FUNCTION_BLOCK WRITE_Manufacturer_label
VAR_INPUT
	Label_In	: ST_Manufacturer_label;
	NodeID		: BYTE; (* This Port No. addresses the CANopen Node (see System Manager) *)	
	Start		: BOOL;
END_VAR
VAR_OUTPUT
	Finished	: BOOL := FALSE;
END_VAR
VAR
	Index		: INT;
	Label		: ST_Manufacturer_label;
	SDO_WRITE 	: FB_SDO_WRITE;
	WriteData		: ARRAY [0..255] OF BYTE;	
	CAN_Objects: INT;
	
	fbTonDelay		: TON;
END_VAR

// Restart after complete run
IF (Index = 255) AND Start THEN
	Index := 0;
END_IF


IF NOT (Index = 255) THEN 
	SDO_WRITE(StartWriting:=FALSE);
	FB_SDO_WRITE_REAL(StartWriting:=FALSE);
END_IF


CASE Index OF	
	0: 
		IF Start THEN	
			Label := Label_In;	
			Finished := FALSE;
			WriteData[0] := DWORD_TO_BYTE(Label.Min_v);
			WriteData[1] := DWORD_TO_BYTE(SHR(Label.Min_v,8));
			WriteData[2] := DWORD_TO_BYTE(SHR(Label.Min_v,16));
			WriteData[3] := DWORD_TO_BYTE(SHR(Label.Min_v,24));		
			SDO_WRITE(	
				AdsNetID		:= GLB.ADSNetID_CAN,
				PortNr			:= 16#1000 + GLB.NodeID,
				CO_Index		:= 16#41C0,
				CO_SubIndex		:= 16#03,
				DataLength		:= 4,
				WriteData		:= WriteData,
				StartWriting	:= TRUE	
			);	
			Index := Index + 1;
		END_IF
	
	
	1: 
		IF SDO_WRITE.WriteDataFinished THEN
			WriteData[0] := DWORD_TO_BYTE(Label.Max_v);
			WriteData[1] := DWORD_TO_BYTE(SHR(Label.Max_v,8));
			WriteData[2] := DWORD_TO_BYTE(SHR(Label.Max_v,16));
			WriteData[3] := DWORD_TO_BYTE(SHR(Label.Max_v,24));		
			SDO_WRITE(	
				AdsNetID		:= GLB.ADSNetID_CAN,
				PortNr			:= 16#1000 + GLB.NodeID,
				CO_Index		:= 16#41C0,
				CO_SubIndex		:= 16#04,
				DataLength		:= 4,
				WriteData		:= WriteData,
				StartWriting	:= TRUE	
			);	
			Index := Index + 1;
		ELSE
			SDO_WRITE();
		END_IF
	
	
	2: 
		IF SDO_WRITE.WriteDataFinished THEN
			WriteData[0] := DWORD_TO_BYTE(Label.Motor_rated_current);
			WriteData[1] := DWORD_TO_BYTE(SHR(Label.Motor_rated_current,8));
			WriteData[2] := DWORD_TO_BYTE(SHR(Label.Motor_rated_current,16));
			WriteData[3] := DWORD_TO_BYTE(SHR(Label.Motor_rated_current,24));		
			SDO_WRITE(	
				AdsNetID		:= GLB.ADSNetID_CAN,
				PortNr			:= 16#1000 + GLB.NodeID,
				CO_Index		:= 16#41C0,
				CO_SubIndex		:= 16#05,
				DataLength		:= 4,
				WriteData		:= WriteData,
				StartWriting	:= TRUE	
			);	
			Index := Index + 1;
		ELSE
			SDO_WRITE();
		END_IF
	
	
	3: 
		IF SDO_WRITE.WriteDataFinished THEN
			WriteData[0] := DWORD_TO_BYTE(Label.Drive_rated_current);
			WriteData[1] := DWORD_TO_BYTE(SHR(Label.Drive_rated_current,8));
			WriteData[2] := DWORD_TO_BYTE(SHR(Label.Drive_rated_current,16));
			WriteData[3] := DWORD_TO_BYTE(SHR(Label.Drive_rated_current,24));		
			SDO_WRITE(	
				AdsNetID		:= GLB.ADSNetID_CAN,
				PortNr			:= 16#1000 + GLB.NodeID,
				CO_Index		:= 16#41C0,
				CO_SubIndex		:= 16#06,
				DataLength		:= 4,
				WriteData		:= WriteData,
				StartWriting	:= TRUE	
			);	
			Index := Index + 1;
		ELSE
			SDO_WRITE();
		END_IF
	
	
	4: 
		IF SDO_WRITE.WriteDataFinished THEN
			WriteData[0] := DWORD_TO_BYTE(Label.Max_current);
			WriteData[1] := DWORD_TO_BYTE(SHR(Label.Max_current,8));
			WriteData[2] := 0;
			WriteData[3] := 0;		
			SDO_WRITE(	
				AdsNetID		:= GLB.ADSNetID_CAN,
				PortNr			:= 16#1000 + GLB.NodeID,
				CO_Index		:= 16#41C0,
				CO_SubIndex		:= 16#07,
				DataLength		:= 2,
				WriteData		:= WriteData,
				StartWriting	:= TRUE	
			);	
			Index := Index + 1;
		ELSE
			SDO_WRITE();
		END_IF	
		
		
	5: 
		IF SDO_WRITE.WriteDataFinished THEN
			WriteData[0] := DWORD_TO_BYTE(Label.Motor_rated_torque);
			WriteData[1] := DWORD_TO_BYTE(SHR(Label.Motor_rated_torque,8));
			WriteData[2] := DWORD_TO_BYTE(SHR(Label.Motor_rated_torque,16));
			WriteData[3] := DWORD_TO_BYTE(SHR(Label.Motor_rated_torque,24));		
			SDO_WRITE(	
				AdsNetID		:= GLB.ADSNetID_CAN,
				PortNr			:= 16#1000 + GLB.NodeID,
				CO_Index		:= 16#41C0,
				CO_SubIndex		:= 16#08,
				DataLength		:= 4,
				WriteData		:= WriteData,
				StartWriting	:= TRUE	
			);	
			Index := Index + 1;
		ELSE
			SDO_WRITE();
		END_IF
	
	
	6: 
		IF SDO_WRITE.WriteDataFinished THEN
			WriteData[0] := DWORD_TO_BYTE(Label.Max_torque);
			WriteData[1] := DWORD_TO_BYTE(SHR(Label.Max_torque,8));
			WriteData[2] := 0;
			WriteData[3] := 0;		
			SDO_WRITE(	
				AdsNetID		:= GLB.ADSNetID_CAN,
				PortNr			:= 16#1000 + GLB.NodeID,
				CO_Index		:= 16#41C0,
				CO_SubIndex		:= 16#09,
				DataLength		:= 2,
				WriteData		:= WriteData,
				StartWriting	:= TRUE	
			);	
			Index := Index + 1;
		ELSE
			SDO_WRITE();
		END_IF
			
		
	7: 
		IF SDO_WRITE.WriteDataFinished THEN
			WriteData[0] := DWORD_TO_BYTE(Label.Motor_rated_speed);
			WriteData[1] := DWORD_TO_BYTE(SHR(Label.Motor_rated_speed,8));
			WriteData[2] := DWORD_TO_BYTE(SHR(Label.Motor_rated_speed,16));
			WriteData[3] := DWORD_TO_BYTE(SHR(Label.Motor_rated_speed,24));		
			SDO_WRITE(	
				AdsNetID		:= GLB.ADSNetID_CAN,
				PortNr			:= 16#1000 + GLB.NodeID,
				CO_Index		:= 16#41C0,
				CO_SubIndex		:= 16#0A,
				DataLength		:= 4,
				WriteData		:= WriteData,
				StartWriting	:= TRUE	
			);	
			Index := Index + 1;
		ELSE
			SDO_WRITE();
		END_IF
	
		
	8: 
		IF SDO_WRITE.WriteDataFinished THEN
			WriteData[0] := DWORD_TO_BYTE(Label.Number_of_pole_pairs);
			WriteData[1] := DWORD_TO_BYTE(SHR(Label.Number_of_pole_pairs,8));
			WriteData[2] := 0;
			WriteData[3] := 0;		
			SDO_WRITE(	
				AdsNetID		:= GLB.ADSNetID_CAN,
				PortNr			:= 16#1000 + GLB.NodeID,
				CO_Index		:= 16#41C0,
				CO_SubIndex		:= 16#0B,
				DataLength		:= 2,
				WriteData		:= WriteData,
				StartWriting	:= TRUE	
			);	
			Index := Index + 1;
		ELSE
			SDO_WRITE();
		END_IF
			
		
	9: 
		IF SDO_WRITE.WriteDataFinished THEN
			FB_SDO_WRITE_REAL(	
				AdsNetID		:= GLB.ADSNetID_CAN,
				PortNr			:= 16#1000 + GLB.NodeID,
				CO_Index		:= 16#41C0,
				CO_SubIndex		:= 16#0C,
				WriteData		:= Label.Motor_torque_constant,
				StartWriting	:= TRUE	
			);	
			Index := Index + 1;
		ELSE
			SDO_WRITE();
		END_IF
			
		
	10: 
		IF FB_SDO_WRITE_REAL.WriteDataFinished THEN
			FB_SDO_WRITE_REAL(	
				AdsNetID		:= GLB.ADSNetID_CAN,
				PortNr			:= 16#1000 + GLB.NodeID,
				CO_Index		:= 16#41C0,
				CO_SubIndex		:= 16#0D,
				WriteData		:= Label.Flux_producing_P_gain,
				StartWriting	:= TRUE	
			);	
			Index := Index + 1;
		ELSE
			FB_SDO_WRITE_REAL();
		END_IF
			
		
	11: 
		IF FB_SDO_WRITE_REAL.WriteDataFinished THEN
			FB_SDO_WRITE_REAL(	
				AdsNetID		:= GLB.ADSNetID_CAN,
				PortNr			:= 16#1000 + GLB.NodeID,
				CO_Index		:= 16#41C0,
				CO_SubIndex		:= 16#0E,
				WriteData		:= Label.Flux_producing_I_gain,
				StartWriting	:= TRUE	
			);	
			Index := Index + 1;
		ELSE
			FB_SDO_WRITE_REAL();
		END_IF
			
		
	12: 
		IF FB_SDO_WRITE_REAL.WriteDataFinished THEN	
			FB_SDO_WRITE_REAL(	
				AdsNetID		:= GLB.ADSNetID_CAN,
				PortNr			:= 16#1000 + GLB.NodeID,
				CO_Index		:= 16#41C0,
				CO_SubIndex		:= 16#0F,
				WriteData		:= Label.Torque_producing_P_gain,
				StartWriting	:= TRUE	
			);	
			Index := Index + 1;
		ELSE
			FB_SDO_WRITE_REAL();
		END_IF
			
		
	13: 
		IF FB_SDO_WRITE_REAL.WriteDataFinished THEN
			FB_SDO_WRITE_REAL(	
				AdsNetID		:= GLB.ADSNetID_CAN,
				PortNr			:= 16#1000 + GLB.NodeID,
				CO_Index		:= 16#41C0,
				CO_SubIndex		:= 16#10,
				WriteData		:= Label.Torque_producing_I_gain,
				StartWriting	:= TRUE	
			);	
			Index := Index + 1;
		ELSE
			FB_SDO_WRITE_REAL();
		END_IF
			
		
	14: 
		IF FB_SDO_WRITE_REAL.WriteDataFinished THEN
			WriteData[0] := DWORD_TO_BYTE(Label.Magnetic_encoder_offset);
			WriteData[1] := DWORD_TO_BYTE(SHR(Label.Magnetic_encoder_offset,8));
			WriteData[2] := 0;
			WriteData[3] := 0;		
			SDO_WRITE(	
				AdsNetID		:= GLB.ADSNetID_CAN,
				PortNr			:= 16#1000 + GLB.NodeID,
				CO_Index		:= 16#41C0,
				CO_SubIndex		:= 16#11,
				DataLength		:= 2,
				WriteData		:= WriteData,
				StartWriting	:= TRUE	
			);	
			Index := Index + 1;
		ELSE
			FB_SDO_WRITE_REAL();
		END_IF
			
		
	15: 
		IF SDO_WRITE.WriteDataFinished THEN
			WriteData[0] := DWORD_TO_BYTE(Label.Motor_with_brake);
			WriteData[1] := DWORD_TO_BYTE(SHR(Label.Motor_with_brake,8));
			WriteData[2] := 0;
			WriteData[3] := 0;		
			SDO_WRITE(	
				AdsNetID		:= GLB.ADSNetID_CAN,
				PortNr			:= 16#1000 + GLB.NodeID,
				CO_Index		:= 16#41C0,
				CO_SubIndex		:= 16#12,
				DataLength		:= 2,
				WriteData		:= WriteData,
				StartWriting	:= TRUE	
			);	
			Index := Index + 1;
		ELSE
			SDO_WRITE();
		END_IF
			
		
	16: 
		IF SDO_WRITE.WriteDataFinished THEN
			WriteData[0] := DWORD_TO_BYTE(Label.Encoder_mode_adjust);
			WriteData[1] := DWORD_TO_BYTE(SHR(Label.Encoder_mode_adjust,8));
			WriteData[2] := 0;
			WriteData[3] := 0;		
			SDO_WRITE(	
				AdsNetID		:= GLB.ADSNetID_CAN,
				PortNr			:= 16#1000 + GLB.NodeID,
				CO_Index		:= 16#41C0,
				CO_SubIndex		:= 16#13,
				DataLength		:= 2,
				WriteData		:= WriteData,
				StartWriting	:= TRUE	
			);	
			Index := Index + 1;
		ELSE
			SDO_WRITE();
		END_IF
			
		
	17: 
		IF SDO_WRITE.WriteDataFinished THEN
			WriteData[0] := DWORD_TO_BYTE(Label.Motor_max_speed);
			WriteData[1] := DWORD_TO_BYTE(SHR(Label.Motor_max_speed,8));
			WriteData[2] := 0;
			WriteData[3] := 0;		
			SDO_WRITE(	
				AdsNetID		:= GLB.ADSNetID_CAN,
				PortNr			:= 16#1000 + GLB.NodeID,
				CO_Index		:= 16#41C0,
				CO_SubIndex		:= 16#14,
				DataLength		:= 2,
				WriteData		:= WriteData,
				StartWriting	:= TRUE	
			);	
			Index := Index + 1;
		ELSE
			SDO_WRITE();
		END_IF
			
		
	18: 
		IF SDO_WRITE.WriteDataFinished THEN
			FB_SDO_WRITE_REAL(	
				AdsNetID		:= GLB.ADSNetID_CAN,
				PortNr			:= 16#1000 + GLB.NodeID,
				CO_Index		:= 16#41C0,
				CO_SubIndex		:= 16#15,
				WriteData		:= Label.Rotor_inertia,
				StartWriting	:= TRUE	
			);	
			Index := Index + 1;
		ELSE
			SDO_WRITE();
		END_IF
			
		
	19: 
		IF FB_SDO_WRITE_REAL.WriteDataFinished THEN		
			FB_SDO_WRITE_REAL(	
				AdsNetID		:= GLB.ADSNetID_CAN,
				PortNr			:= 16#1000 + GLB.NodeID,
				CO_Index		:= 16#41C0,
				CO_SubIndex		:= 16#17,
				WriteData		:= Label.Motor_time_at_peak,
				StartWriting	:= TRUE	
			);	
			Index := Index + 1;
		ELSE
			FB_SDO_WRITE_REAL();
		END_IF
			
		
	20: 
		IF FB_SDO_WRITE_REAL.WriteDataFinished THEN		
			FB_SDO_WRITE_REAL(	
				AdsNetID		:= GLB.ADSNetID_CAN,
				PortNr			:= 16#1000 + GLB.NodeID,
				CO_Index		:= 16#41C0,
				CO_SubIndex		:= 16#18,
				WriteData		:= Label.Drive_time_at_peak,
				StartWriting	:= TRUE	
			);	
			Index := Index + 1;
		ELSE
			FB_SDO_WRITE_REAL();
		END_IF
			
		
	21: 
		IF FB_SDO_WRITE_REAL.WriteDataFinished THEN
			WriteData[0] := Label.Singleturn_resolution;
			WriteData[1] := 0;
			WriteData[2] := 0;
			WriteData[3] := 0;			
			SDO_WRITE(	
				AdsNetID		:= GLB.ADSNetID_CAN,
				PortNr			:= 16#1000 + GLB.NodeID,
				CO_Index		:= 16#41C0,
				CO_SubIndex		:= 16#19,
				DataLength		:= 1,
				WriteData		:= WriteData,
				StartWriting	:= TRUE	
			);	
			Index := Index + 1;
		ELSE
			FB_SDO_WRITE_REAL();
		END_IF
			
		
	22: 
		IF SDO_WRITE.WriteDataFinished THEN
			WriteData[0] := Label.Multiturn_resolution;
			WriteData[1] := 0;
			WriteData[2] := 0;
			WriteData[3] := 0;		
			SDO_WRITE(	
				AdsNetID		:= GLB.ADSNetID_CAN,
				PortNr			:= 16#1000 + GLB.NodeID,
				CO_Index		:= 16#41C0,
				CO_SubIndex		:= 16#1A,
				DataLength		:= 1,
				WriteData		:= WriteData,
				StartWriting	:= TRUE	
			);	
			Index := Index + 1;
		ELSE
			SDO_WRITE();
		END_IF
		
	
	23: // SAVE
		IF SDO_WRITE.WriteDataFinished THEN
			WriteData[0] := 0;
			WriteData[1] := 0;
			WriteData[2] := 0;
			WriteData[3] := 0;		
			SDO_WRITE(	
				AdsNetID		:= GLB.ADSNetID_CAN,
				PortNr			:= 16#1000 + GLB.NodeID,
				CO_Index		:= 16#1010,
				CO_SubIndex		:= 16#4,
				DataLength		:= 4,
				WriteData		:= WriteData,
				StartWriting	:= TRUE	
			);	
			Index := Index + 1;
		ELSE
			SDO_WRITE();
		END_IF		
			
			
	24: // Wait 500 ms for save process
		fbTonDelay(IN := TRUE, PT:= T#500MS);
		IF fbTonDelay.Q THEN
			fbTonDelay(IN := FALSE);
			Index := Index + 1;	
		END_IF
		
		
	255: // Finished 
		Finished := TRUE;
			
		
	ELSE
		Index := 255;
	
END_CASE

END_FUNCTION_BLOCK

(* stored: Version 1.1.0.1, ProductVersion 3.1.4024.11
   POU WRITE_Manufacturer_label: Id {70da4c45-a45c-433d-9aa9-64e7022830d4}, SpecialFunc None *)
